Fanuc KAREL source: kb00021.compact.KL

PROGRAM KB00021
%STACKSIZE=65535
%PRIORITY=65535
%NOLOCKGROUP
VAR
P1 : STRING[80]
P2 : INTEGER
BEGIN
P1='A'
P2=1
CLEAR(P1,P2)
END KB00021
